INTERFACE itfActuate

METHOD mTurnOffAuto : BOOL
VAR_INPUT
END_VAR
END_METHOD

METHOD mTurnOffManual : BOOL
VAR_INPUT
END_VAR
END_METHOD

METHOD mTurnOnAuto : BOOL
VAR_INPUT
END_VAR
END_METHOD

METHOD mTurnOnManual : BOOL
VAR_INPUT
END_VAR
END_METHOD

PROPERTY pCoil : Bool
GET
END_GET
SET
END_SET
END_PROPERTY

PROPERTY pStart : Bool
GET
END_GET
SET
END_SET
END_PROPERTY

PROPERTY pStop : Bool
GET
END_GET
SET
END_SET
END_PROPERTY

END_INTERFACE

(* stored: Version 1.1.0.1, ProductVersion 3.1.4024.12
   Itf itfActuate: Id {c27dcbc9-0a44-4669-9d91-356bb6a085b8}
   Method mTurnOffAuto: Id {11785087-ff94-402d-92d0-da83ce6aa0a9}
   Method mTurnOffManual: Id {915c598e-e075-4fe6-a9db-78c85df4f985}
   Method mTurnOnAuto: Id {4d358000-52e8-4f72-a58a-e5e326555f83}
   Method mTurnOnManual: Id {06d9b11e-9a2a-4bf1-a6e2-f2f711951ae0}
   Property pCoil: Id {f8e9c5d9-6d59-404a-8c24-9242cb1e5395}
   Get Get: Id {755145f7-d13b-4442-8ea6-3b290e7993ff}
   Set Set: Id {e900090f-35ce-452f-a9f1-a775a3fb26ec}
   Property pStart: Id {a1af4811-f7c9-4081-b328-459541259638}
   Get Get: Id {5906180f-bb6c-4635-a64f-40dc50e81fb2}
   Set Set: Id {b7dd49f8-f8f4-4a4b-8e8c-a5510b1f3fdd}
   Property pStop: Id {34f9b22d-fdc5-4373-9d58-2864878d6f10}
   Get Get: Id {6fbea6b1-7592-4268-9fa7-ef9ac49f96c1}
   Set Set: Id {0b8b9186-9983-422b-9162-694e5012e86b} *)
